LAYER IOs
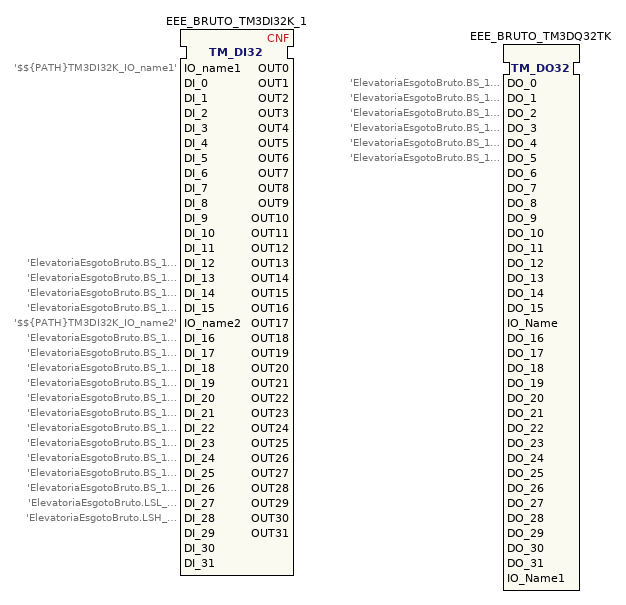
  (* EEE_BRUTO *)
  FBS
    EEE_BRUTO_TM3DI32K_1 : TM_DI32(IO_name1 := '$${PATH}TM3DI32K_IO_name1', IO_name2 := '$${PATH}TM3DI32K_IO_name2', DI_12 := 'ElevatoriaEsgotoBruto.BS_100_01.stsLocal', DI_13 := 'ElevatoriaEsgotoBruto.BS_100_01.stsRemoto', DI_14 := 'ElevatoriaEsgotoBruto.BS_100_01.stsLigado', DI_15 := 'ElevatoriaEsgotoBruto.BS_100_01.stsSemFalha', DI_16 := 'ElevatoriaEsgotoBruto.BS_100_01.stsProtecaoTermica', DI_17 := 'ElevatoriaEsgotoBruto.BS_100_02.stsLocal', DI_18 := 'ElevatoriaEsgotoBruto.BS_100_02.stsRemoto', DI_19 := 'ElevatoriaEsgotoBruto.BS_100_02.stsLigado', DI_20 := 'ElevatoriaEsgotoBruto.BS_100_02.stsSemFalha', DI_21 := 'ElevatoriaEsgotoBruto.BS_100_02.stsProtecaoTermica', DI_22 := 'ElevatoriaEsgotoBruto.BS_100_03.stsLocal', DI_23 := 'ElevatoriaEsgotoBruto.BS_100_03.stsRemoto', DI_24 := 'ElevatoriaEsgotoBruto.BS_100_03.stsLigado', DI_25 := 'ElevatoriaEsgotoBruto.BS_100_03.stsSemFalha', DI_26 := 'ElevatoriaEsgotoBruto.BS_100_03.stsProtecaoTermica', DI_27 := 'ElevatoriaEsgotoBruto.LSL_100_04.stsBoiaAtiva', DI_28 := 'ElevatoriaEsgotoBruto.LSH_100_05.stsBoiaAtiva');
    EEE_BRUTO_TM3DQ32TK : TM_DO32(DO_0 := 'ElevatoriaEsgotoBruto.BS_100_01.cmdAcionamento', DO_1 := 'ElevatoriaEsgotoBruto.BS_100_01.cmdReset', DO_2 := 'ElevatoriaEsgotoBruto.BS_100_02.cmdAcionamento', DO_3 := 'ElevatoriaEsgotoBruto.BS_100_02.cmdReset', DO_4 := 'ElevatoriaEsgotoBruto.BS_100_03.cmdAcionamento', DO_5 := 'ElevatoriaEsgotoBruto.BS_100_03.cmdReset');
  END_FBS
END_LAYER
